// TwinCAT 3 PLC project PixelLEDComponentLib
// ProgramVersion: 3.1.4024.0
// libraries:
//   SPT Base Types, * (Beckhoff Automation LLC)
//   Tc2_Standard, * (Beckhoff Automation GmbH)
//   Tc2_System, * (Beckhoff Automation GmbH)
//   Tc3_Module, * (Beckhoff Automation GmbH)
// project tree:
//   PixelColourObjects/ ColourOptions.TcDUT, ColourPallette.TcPOU
//   PixelStreamClass/ PixelStreamClass.TcPOU
//   PixelVideoObjects/ ITF_Video.TcIO, PixelVideoClass.TcPOU
//   PixelWritterObjects/ Colour.TcDUT, Command.TcDUT, Control.TcDUT, ExtendedCommand.TcDUT, ExtendedControl.TcDUT, ITF_PixelWritter.TcIO, PixelWritter.TcPOU, Status.TcDUT
//   / PlcTask.TcTTO
//   POUs/ MAIN.TcPOU

CONFIGURATION PixelLEDComponentLib
    RESOURCE PLC ON TwinCAT3
        TASK PlcTask(INTERVAL := T#10ms, PRIORITY := 20);
        PROGRAM MAIN WITH PlcTask : MAIN;
    END_RESOURCE
END_CONFIGURATION

// ---- PixelColourObjects/ColourOptions.TcDUT
{attribute 'qualified_only' := ''}
{attribute 'strict' := ''}
TYPE ColourOptions :
(
	DARK_RED := 0,
	CRIMSON := 3,
	RED := 4,
	TOMATO := 5,
	SALMON := 10,
	DARK_ORANGE := 13,
	ORANGE := 14,
	GOLD := 15,
	GOLDEN_ROD := 17,
	DARK_KHAKI := 19,
	OLIVE := 21,
	YELLOW := 22,
	LAWN_GREEN := 26,
	GREEN := 30,
	FOREST_GREEN := 31,
	LIME := 32,
	LIGHT_SEA_GREEN := 42,
	TEAL := 44,
	AQUA := 46,
	TURQUOISE := 50,
	STEEL_BLUE := 56,
	DEEP_SKY_BLUE := 58,
	NAVY := 64,
	BLUE := 67,
	BLUE_VIOLET := 69,
	MEDIUM_PURPLE := 74,
	PURPLE := 79,
	MAGENTA := 83,
	DEEP_PINK := 87,
	HOT_PINK := 90,
	LEMON_CHIFFON := 97,
	SADDLE_BROWN := 100,
	SANDY_BROWN := 104,
	MOCCASIN := 108,
	MINT_CREAM := 117,
	SLATE_GREY := 118,
	LAVENDER := 121,
	BLACK := 129,
	GREY := 131,
	SILVER := 133,
	WHITE := 137
);
END_TYPE

// ---- PixelWritterObjects/Colour.TcDUT
TYPE Colour :
STRUCT
	Red: USINT;
	Green: USINT;
	Blue: USINT;
END_STRUCT
END_TYPE

// ---- PixelWritterObjects/Command.TcDUT
TYPE Command :
STRUCT
	Command: USINT;
	Index: UINT;
	Length: UINT;
	Parameter: UINT;
	Colours: Colour;
END_STRUCT
END_TYPE

// ---- PixelWritterObjects/Control.TcDUT
TYPE Control :
STRUCT
	Execute: BOOL;
	Send: BOOL;
	Update: BOOL;
	PixelCommand: Command;
END_STRUCT
END_TYPE

// ---- PixelWritterObjects/ExtendedCommand.TcDUT
TYPE ExtendedCommand :
STRUCT
	Index: USINT;
	Segment: ARRAY[0..7] OF UDINT;
END_STRUCT
END_TYPE

// ---- PixelWritterObjects/ExtendedControl.TcDUT
TYPE ExtendedControl :
STRUCT
	Execute: BOOL;
	Send: BOOL;
	Update: BOOL;
	Write: BOOL;
	Command: ExtendedCommand;
END_STRUCT
END_TYPE

// ---- PixelWritterObjects/Status.TcDUT
TYPE Status :
STRUCT
	Busy: BOOL;
	Transmit: BOOL;
	SendAck: BOOL;
	UpdateAck: BOOL;
	CommandAck: BOOL;
	CommandReject: BOOL;
	Warning: BOOL;
	Error: BOOL;
END_STRUCT
END_TYPE

// ---- PixelVideoObjects/ITF_Video.TcIO
INTERFACE ITF_Video

METHOD GetNextFrame : ARRAY[0..255] OF UDINT
END_METHOD

END_INTERFACE

// ---- PixelWritterObjects/ITF_PixelWritter.TcIO
INTERFACE ITF_PixelWritter

METHOD ClearPixelArrayCommand : BOOL
END_METHOD

METHOD ForwardCommandToFrameBuffer : BOOL
END_METHOD

METHOD ForwardExtCommandToFrame : BOOL
END_METHOD

METHOD SendCommandToPixelBuffer : BOOL
VAR_INPUT
	NewCommand: Command;
END_VAR
END_METHOD

METHOD SendExtCommand : BOOL
VAR_INPUT
	NewCommand: ExtendedCommand;
END_VAR
END_METHOD

END_INTERFACE

// ---- POUs/MAIN.TcPOU
PROGRAM MAIN
VAR
	EL2574Control : PixelWritter;
	MyVideo : PixelVideoClass;
	FilmControl : PixelStreamClass;
	MyCommand : Command;
	MyColourPallette : ColourPallette;
	MyColour : ColourOptions;
	init: BOOL;
	SendManualCommand : BOOL;
	SendManualUpdate : BOOL;
	SendClearCommand : BOOL;
END_VAR

IF NOT init THEN
	FilmControl.RegisterAVideo(MyVideo := MyVideo);
	FilmControl.RegisterMyPixelArray(MYPixelWritter := EL2574Control);
	init := TRUE;
END_IF
FilmControl.CyclicLogic();
EL2574Control.CyclicLogic();


MyCommand.Colours := MyColourPallette.GetColourComponents(Colour := MyColour);
IF SendManualCommand THEN
	EL2574Control.SendCommandToPixelBuffer(NewCommand := MyCommand);
	SendManualCommand := FALSE;
END_IF
IF SendManualUpdate THEN
	EL2574Control.ForwardCommandToFrameBuffer();
	SendManualUpdate := FALSE;
END_IF
IF SendClearCommand THEN
	EL2574Control.ClearPixelArrayCommand();
	SendClearCommand := FALSE;
END_IF

END_PROGRAM

// ---- PixelWritterObjects/PixelWritter.TcPOU
FUNCTION_BLOCK PixelWritter EXTENDS FB_ComponentBase IMPLEMENTS ITF_PixelWritter
VAR
	CtrlOut AT %Q*: Control;
	StatusIn AT %I*: Status;
	ExtCtrlOut AT %Q*: ExtendedControl;
	UpdateRTrig: R_TRIG;
	UpdateFTrig: F_TRIG;
	ClearPixels: BOOL;
END_VAR

METHOD ClearPixelArrayCommand : BOOL
IF NOT ClearPixels THEN
	CtrlOut.PixelCommand.Command := 2;
	CtrlOut.Execute := NOT CtrlOut.Execute;
END_IF
END_METHOD

METHOD CyclicLogic
SUPER^.CyclicLogic();
UpdateFTrig(CLK := StatusIn.UpdateAck);
UpdateRTrig(CLK := StatusIn.UpdateAck);
IF UpdateFTrig.Q OR UpdateRTrig.Q THEN
	CtrlOut.Update := FALSE;
	ExtCtrlOut.Update := FALSE;
END_IF
END_METHOD

METHOD ForwardCommandToFrameBuffer : BOOL
IF NOT ForwardCommandToFrameBuffer THEN
	CtrlOut.Execute := NOT CtrlOut.Execute;
	CtrlOut.Update := TRUE;
	ForwardCommandToFrameBuffer := TRUE;
END_IF
END_METHOD

METHOD ForwardExtCommandToFrame : BOOL
IF NOT ForwardExtCommandToFrame THEN
	ExtCtrlOut.Execute := NOT ExtCtrlOut.Execute;
	ExtCtrlOut.Update := TRUE;
	ExtCtrlOut.Write := FALSE;
	ForwardExtCommandToFrame := TRUE;
END_IF
END_METHOD

METHOD SendCommandToPixelBuffer : BOOL
VAR_INPUT
	NewCommand: Command;
END_VAR
IF NOT StatusIn.Busy THEN
	SendCommandToPixelBuffer := TRUE;
	CtrlOut.PixelCommand := NewCommand;
	CtrlOut.Execute := NOT CtrlOut.Execute;
END_IF
END_METHOD

METHOD SendExtCommand : BOOL
VAR_INPUT
	NewCommand: ExtendedCommand;
END_VAR
IF NOT StatusIn.Busy THEN
	SendExtCommand := TRUE;
	ExtCtrlOut.Command := NewCommand;
	ExtCtrlOut.Write := TRUE;
	ExtCtrlOut.Execute := NOT ExtCtrlOut.Execute;
END_IF
END_METHOD

END_FUNCTION_BLOCK

// ---- PixelVideoObjects/PixelVideoClass.TcPOU
FUNCTION_BLOCK PixelVideoClass EXTENDS FB_ComponentBase IMPLEMENTS ITF_Video
VAR
	CurrentFrame: INT := 0;
	TotalFramesInFilm: INT;
	ThisVideo: ARRAY[0..99, 0..255] OF UDINT;
	I: INT;
END_VAR

METHOD PUBLIC  CyclicLogic
VAR_INPUT
END_VAR
SUPER^.CyclicLogic();
END_METHOD

METHOD GetNextFrame : ARRAY[0..255] OF UDINT
FOR I := 0 TO 255 DO
	GetNextFrame[I] := ThisVideo[CurrentFrame,I];
END_FOR

IF CurrentFrame = TotalFramesInFilm - 1 THEN
	CurrentFrame := 0;
ELSE
	CurrentFrame := CurrentFrame + 1;
END_IF
END_METHOD

END_FUNCTION_BLOCK

// ---- PixelStreamClass/PixelStreamClass.TcPOU
FUNCTION_BLOCK PixelStreamClass EXTENDS FB_ComponentBase
VAR
	_PixelWriter: ITF_PixelWritter;
	_Video: ITF_Video;
	State: INT;
	Play: BOOL;
	currentFrame: ARRAY[0..255] OF UDINT;
	NewCommand: ExtendedCommand;
	FrameTimeDelay: TON := (PT := TIME#100ms);
END_VAR

METHOD CyclicLogic
SUPER^.CyclicLogic();

CASE State OF
	0:
		IF Play THEN
			State := 1;
		END_IF
	1:
	    currentFrame :=	_Video.GetNextFrame();
		State := 2;
	2:
		CASE NewCommand.Index OF 
			0,1,4,5,8,9,12,13,16,17,20,21,24,25,28,29:
				NewCommand.Segment[0] := currentFrame[NewCommand.Index * 8 + 0];
				NewCommand.Segment[1] := currentFrame[NewCommand.Index * 8 + 1];
				NewCommand.Segment[2] := currentFrame[NewCommand.Index * 8 + 2];
				NewCommand.Segment[3] := currentFrame[NewCommand.Index * 8 + 3];
				NewCommand.Segment[4] := currentFrame[NewCommand.Index * 8 + 4];
				NewCommand.Segment[5] := currentFrame[NewCommand.Index * 8 + 5];
				NewCommand.Segment[6] := currentFrame[NewCommand.Index * 8 + 6];
				NewCommand.Segment[7] := currentFrame[NewCommand.Index * 8 + 7];
			2,6,10,14,18,22,26,30:
				NewCommand.Segment[7] := currentFrame[(NewCommand.Index + 1) * 8 + 0];
				NewCommand.Segment[6] := currentFrame[(NewCommand.Index + 1) * 8 + 1];
				NewCommand.Segment[5] := currentFrame[(NewCommand.Index + 1) * 8 + 2];
				NewCommand.Segment[4] := currentFrame[(NewCommand.Index + 1) * 8 + 3];
				NewCommand.Segment[3] := currentFrame[(NewCommand.Index + 1) * 8 + 4];
				NewCommand.Segment[2] := currentFrame[(NewCommand.Index + 1) * 8 + 5];
				NewCommand.Segment[1] := currentFrame[(NewCommand.Index + 1) * 8 + 6];
				NewCommand.Segment[0] := currentFrame[(NewCommand.Index + 1) * 8 + 7];
			3,7,11,15,19,23,27,31:
				NewCommand.Segment[7] := currentFrame[(NewCommand.Index - 1) * 8 + 0];
				NewCommand.Segment[6] := currentFrame[(NewCommand.Index - 1) * 8 + 1];
				NewCommand.Segment[5] := currentFrame[(NewCommand.Index - 1) * 8 + 2];
				NewCommand.Segment[4] := currentFrame[(NewCommand.Index - 1) * 8 + 3];
				NewCommand.Segment[3] := currentFrame[(NewCommand.Index - 1) * 8 + 4];
				NewCommand.Segment[2] := currentFrame[(NewCommand.Index - 1) * 8 + 5];
				NewCommand.Segment[1] := currentFrame[(NewCommand.Index - 1) * 8 + 6];
				NewCommand.Segment[0] := currentFrame[(NewCommand.Index - 1) * 8 + 7];
		END_CASE
		
		State := 3;
	3:
		IF _PixelWriter.SendExtCommand(NewCommand := NewCommand) THEN
			NewCommand.Index := NewCommand.Index + 1;
			IF NewCommand.Index = 32 THEN
				State := 4;
				NewCommand.Index := 0;
			ELSE
				State := 2;
			END_IF
		END_IF
		
	4:
		IF _PixelWriter.ForwardExtCommandToFrame() THEN
			FrameTimeDelay.IN := TRUE;
			State := 5;
		END_IF
	
	5:
		IF FrameTimeDelay.Q THEN
			FrameTimeDelay.IN := FALSE;
			State := 0;
		END_IF
END_CASE

FrameTimeDelay();
END_METHOD

METHOD PlayVideo : BOOL
Play := PlayVideo := TRUE;
END_METHOD

METHOD RegisterAVideo : BOOL
VAR_INPUT
	MyVideo: ITF_Video;
END_VAR
IF _Video = 0 THEN
	_Video := MyVideo;
	RegisterAVideo := true;
END_IF
END_METHOD

METHOD RegisterMyPixelArray : BOOL
VAR_INPUT
	MYPixelWritter: ITF_PixelWritter;
END_VAR
IF _PixelWriter = 0 THEN
	_PixelWriter := MYPixelWritter;
	RegisterMyPixelArray := TRUE;
END_IF
END_METHOD

METHOD StopVideo : BOOL
Play := FALSE;
StopVideo := TRUE;
END_METHOD

END_FUNCTION_BLOCK

// ---- PixelColourObjects/ColourPallette.TcPOU
FUNCTION_BLOCK ColourPallette EXTENDS FB_ComponentBase
VAR
	ColourOptions: ARRAY[0..137] OF Colour := [(Red := 16#8B, Green := 16#0, Blue := 16#0), (Red := 16#0, Green := 16#0, Blue := 16#0), (Red := 16#0, Green := 16#0, Blue := 16#0), (Red := 16#DC, Green := 16#14, Blue := 16#3C), (Red := 16#FF, Green := 16#0, Blue := 16#0), (Red := 16#FF, Green := 16#63, Blue := 16#47), (Red := 16#0, Green := 16#0, Blue := 16#0), (Red := 16#0, Green := 16#0, Blue := 16#0), (Red := 16#0, Green := 16#0, Blue := 16#0), (Red := 16#0, Green := 16#0, Blue := 16#0), (Red := 16#FA, Green := 16#80, Blue := 16#72), (Red := 16#0, Green := 16#0, Blue := 16#0), (Red := 16#0, Green := 16#0, Blue := 16#0), (Red := 16#FF, Green := 16#8C, Blue := 16#0), (Red := 16#FF, Green := 16#A5, Blue := 16#0), (Red := 16#FF, Green := 16#D7, Blue := 16#0), (Red := 16#0, Green := 16#0, Blue := 16#0), (Red := 16#DA, Green := 16#A5, Blue := 16#20), (Red := 16#0, Green := 16#0, Blue := 16#0), (Red := 16#BD, Green := 16#B7, Blue := 16#6B), (Red := 16#0, Green := 16#0, Blue := 16#0), (Red := 16#80, Green := 16#80, Blue := 16#0), (Red := 16#FF, Green := 16#FF, Blue := 16#0), (Red := 16#0, Green := 16#0, Blue := 16#0), (Red := 16#0, Green := 16#0, Blue := 16#0), (Red := 16#0, Green := 16#0, Blue := 16#0), (Red := 16#7C, Green := 16#FC, Blue := 16#0), (Red := 16#0, Green := 16#0, Blue := 16#0), (Red := 16#0, Green := 16#0, Blue := 16#0), (Red := 16#0, Green := 16#0, Blue := 16#0), (Red := 16#0, Green := 16#80, Blue := 16#0), (Red := 16#22, Green := 16#8B, Blue := 16#22), (Red := 16#0, Green := 16#FF, Blue := 16#0), (Red := 16#0, Green := 16#0, Blue := 16#0), (Red := 16#0, Green := 16#0, Blue := 16#0), (Red := 16#0, Green := 16#0, Blue := 16#0), (Red := 16#0, Green := 16#0, Blue := 16#0), (Red := 16#0, Green := 16#0, Blue := 16#0), (Red := 16#0, Green := 16#0, Blue := 16#0), (Red := 16#0, Green := 16#0, Blue := 16#0), (Red := 16#0, Green := 16#0, Blue := 16#0), (Red := 16#0, Green := 16#0, Blue := 16#0), (Red := 16#20, Green := 16#BA, Blue := 16#AA), (Red := 16#0, Green := 16#0, Blue := 16#0), (Red := 16#0, Green := 16#80, Blue := 16#80), (Red := 16#0, Green := 16#0, Blue := 16#0), (Red := 16#0, Green := 16#FF, Blue := 16#FF), (Red := 16#0, Green := 16#0, Blue := 16#0), (Red := 16#0, Green := 16#0, Blue := 16#0), (Red := 16#0, Green := 16#0, Blue := 16#0), (Red := 16#40, Green := 16#E0, Blue := 16#D0), (Red := 16#0, Green := 16#0, Blue := 16#0), (Red := 16#0, Green := 16#0, Blue := 16#0), (Red := 16#0, Green := 16#0, Blue := 16#0), (Red := 16#0, Green := 16#0, Blue := 16#0), (Red := 16#0, Green := 16#0, Blue := 16#0), (Red := 16#46, Green := 16#82, Blue := 16#B4), (Red := 16#0, Green := 16#0, Blue := 16#0), (Red := 16#0, Green := 16#BF, Blue := 16#FF), (Red := 16#0, Green := 16#0, Blue := 16#0), (Red := 16#0, Green := 16#0, Blue := 16#0), (Red := 16#0, Green := 16#0, Blue := 16#0), (Red := 16#0, Green := 16#0, Blue := 16#0), (Red := 16#0, Green := 16#0, Blue := 16#0), (Red := 16#0, Green := 16#0, Blue := 16#80), (Red := 16#0, Green := 16#0, Blue := 16#0), (Red := 16#0, Green := 16#0, Blue := 16#0), (Red := 16#0, Green := 16#0, Blue := 16#FF), (Red := 16#0, Green := 16#0, Blue := 16#0), (Red := 16#8A, Green := 16#2B, Blue := 16#E2), (Red := 16#0, Green := 16#0, Blue := 16#0), (Red := 16#0, Green := 16#0, Blue := 16#0), (Red := 16#0, Green := 16#0, Blue := 16#0), (Red := 16#0, Green := 16#0, Blue := 16#0), (Red := 16#93, Green := 16#70, Blue := 16#DB), (Red := 16#0, Green := 16#0, Blue := 16#0), (Red := 16#0, Green := 16#0, Blue := 16#0), (Red := 16#0, Green := 16#0, Blue := 16#0), (Red := 16#0, Green := 16#0, Blue := 16#0), (Red := 16#80, Green := 16#0, Blue := 16#80), (Red := 16#0, Green := 16#0, Blue := 16#0), (Red := 16#0, Green := 16#0, Blue := 16#0), (Red := 16#0, Green := 16#0, Blue := 16#0), (Red := 16#FF, Green := 16#0, Blue := 16#FF), (Red := 16#0, Green := 16#0, Blue := 16#0), (Red := 16#0, Green := 16#0, Blue := 16#0), (Red := 16#0, Green := 16#0, Blue := 16#0), (Red := 16#FF, Green := 16#14, Blue := 16#93), (Red := 16#0, Green := 16#0, Blue := 16#0), (Red := 16#0, Green := 16#0, Blue := 16#0), (Red := 16#FF, Green := 16#69, Blue := 16#B4), (Red := 16#0, Green := 16#0, Blue := 16#0), (Red := 16#0, Green := 16#0, Blue := 16#0), (Red := 16#0, Green := 16#0, Blue := 16#0), (Red := 16#0, Green := 16#0, Blue := 16#0), (Red := 16#0, Green := 16#0, Blue := 16#0), (Red := 16#0, Green := 16#0, Blue := 16#0), (Red := 16#FF, Green := 16#FA, Blue := 16#CD), (Red := 16#0, Green := 16#0, Blue := 16#0), (Red := 16#0, Green := 16#0, Blue := 16#0), (Red := 16#8B, Green := 16#45, Blue := 16#13), (Red := 16#0, Green := 16#0, Blue := 16#0), (Red := 16#0, Green := 16#0, Blue := 16#0), (Red := 16#0, Green := 16#0, Blue := 16#0), (Red := 16#F4, Green := 16#A4, Blue := 16#60), (Red := 16#0, Green := 16#0, Blue := 16#0), (Red := 16#0, Green := 16#0, Blue := 16#0), (Red := 16#0, Green := 16#0, Blue := 16#0), (Red := 16#FF, Green := 16#E4, Blue := 16#B5), (Red := 16#0, Green := 16#0, Blue := 16#0), (Red := 16#0, Green := 16#0, Blue := 16#0), (Red := 16#0, Green := 16#0, Blue := 16#0), (Red := 16#0, Green := 16#0, Blue := 16#0), (Red := 16#0, Green := 16#0, Blue := 16#0), (Red := 16#0, Green := 16#0, Blue := 16#0), (Red := 16#0, Green := 16#0, Blue := 16#0), (Red := 16#0, Green := 16#0, Blue := 16#0), (Red := 16#F5, Green := 16#FF, Blue := 16#FA), (Red := 16#70, Green := 16#80, Blue := 16#90), (Red := 16#0, Green := 16#0, Blue := 16#0), (Red := 16#0, Green := 16#0, Blue := 16#0), (Red := 16#E6, Green := 16#E6, Blue := 16#FA), (Red := 16#0, Green := 16#0, Blue := 16#0), (Red := 16#0, Green := 16#0, Blue := 16#0), (Red := 16#0, Green := 16#0, Blue := 16#0), (Red := 16#0, Green := 16#0, Blue := 16#0), (Red := 16#0, Green := 16#0, Blue := 16#0), (Red := 16#0, Green := 16#0, Blue := 16#0), (Red := 16#0, Green := 16#0, Blue := 16#0), (Red := 16#0, Green := 16#0, Blue := 16#0), (Red := 16#0, Green := 16#0, Blue := 16#0), (Red := 16#80, Green := 16#80, Blue := 16#80), (Red := 16#0, Green := 16#0, Blue := 16#0), (Red := 16#C0, Green := 16#C0, Blue := 16#C0), (Red := 16#0, Green := 16#0, Blue := 16#0), (Red := 16#0, Green := 16#0, Blue := 16#0), (Red := 16#0, Green := 16#0, Blue := 16#0), (Red := 16#FF, Green := 16#FF, Blue := 16#FF)];
END_VAR

METHOD GetColourComponents : Colour
VAR_INPUT
	Colour: ColourOptions;
END_VAR
GetColourComponents := ColourOptions[Colour];
END_METHOD

END_FUNCTION_BLOCK
